Fanuc KAREL source: NC0052.KL

-- PROVISIONAL review KL for V940-1; original PC SHA256 6f3e186a13fa9b2ea7fee10ceda56bcfcce3ff27f043303465024bd4401a2d9b
-- Incomplete behavior may be omitted. Consult companion uncertainty JSON. Do not deploy.
PROGRAM NC0052
%NOLOCKGROUP
-- UNRESOLVED_LOCAL_POOL 1 cells at code offset 3; source declarations unknown
-- DIRECT_LOCAL_WORD_ACCESS alone does not prove INTEGER, REAL, or BOOLEAN
BEGIN
  -- UNRESOLVED_PC offsets 0-8; opcodes 2B,2C,7B
  -- UNRESOLVED_PC offsets 13-20; opcodes 9D,23
  -- UNRESOLVED_PC offsets 25-42; opcodes 21,40,41,42
  -- UNRESOLVED_PC offsets 47-81; opcodes 21,2E,52,23,7A,40,41,42
  -- UNRESOLVED_PC offsets 86-110; opcodes 21,2E,52,23,7A,43
  -- UNRESOLVED_PC offsets 115-129; opcodes 21,9D,52,23
  -- UNRESOLVED_PC offsets 139-143; opcodes 7F
  -- UNRESOLVED_PC offsets 148-152; opcodes 27,AA
  -- UNRESOLVED_PC offsets 157-161; opcodes 7F
END NC0052
